Staubli VAL3: endCycle.pgx

public program endCycle()
  local num i
  local string message
begin
  cycleStatus:bToEnd=true
  watch(cycleStatus:bToEnd==false,1)
end
